(* IEC 61131-3 sources: volt/packages/volt-lsp-iec/test-corpus/pro2193/Device/Plc Logic/Application/99 Library/Function Blocks/Sensors, 4 files *)

(* ---- DigitalSensorFB.pou ---- *)
// Basic FB for a digital sensor, adds invert functionality
{attribute 'no_explicit_call' := 'No need to call this FB. No code to execute!'}
{attribute 'symbol' := 'none'}
{attribute 'monitoring_display' := 'IsActive'}
FUNCTION_BLOCK DigitalSensorFB
IMPLEMENTS IDigitalSensor
VAR_INPUT
	{attribute 'symbol' := 'read'}		sensorInput		: BOOL;
END_VAR
VAR
	_isInverted		: BOOL;
END_VAR

%LANGUAGE ST

END_FUNCTION_BLOCK

// FB_Init is always available implicitly and it is used primarily for initialization.
// The return value is not evaluated. For a specific influence, you can also declare the
// methods explicitly and provide additional code there with the standard initialization
// code. You can evaluate the return value.
{attribute 'hide'}
METHOD FB_Init: BOOL
VAR_INPUT
	bInitRetains: BOOL; // TRUE: the retain variables are initialized (reset warm / reset cold)
	bInCopyCode: BOOL;  // TRUE: the instance will be copied to the copy code afterward (online change)

	invert			: BOOL;	// Sensor or photocell signal should be inverted
END_VAR

%LANGUAGE ST
_isInverted := invert;

END_METHOD

// Sensor is active (SensorInput is opposite of the Invert signal)
{attribute 'monitoring':='call'}
PROPERTY IsActive : BOOL

GET
PUBLIC
VAR
END_VAR

%LANGUAGE ST
IsActive := SensorInput = NOT _isInverted;

END_GET
END_PROPERTY

// Sensor is inactive (SensorInput is false (or true when inverted))
{attribute 'monitoring':='call'}
PROPERTY IsInactive : BOOL

GET
PUBLIC
VAR
END_VAR

%LANGUAGE ST
IsInactive := NOT IsActive;

END_GET
END_PROPERTY

(* ---- DigitalSensorWithEnableFB.pou ---- *)
// When disabled a sensor will always return TRUE when asked! So the program will continue and ignore the sensor.
{attribute 'no_explicit_call' := 'No need to call this FB. No code to execute!'}
{attribute 'symbol' := 'none'}
{attribute 'monitoring_display' := 'IsActive'}
FUNCTION_BLOCK DigitalSensorWithEnableFB
EXTENDS DigitalSensorFB
VAR
	_isEnabled		: BOOL;
END_VAR

%LANGUAGE ST

END_FUNCTION_BLOCK

// Sensor is active (SensorInput is opposite of the Invert signal)
{attribute 'monitoring':='call'}
PROPERTY IsActive : BOOL

GET
PUBLIC
VAR
END_VAR

%LANGUAGE ST
IsActive := NOT IsEnabled OR_ELSE SUPER^.IsActive;

END_GET
END_PROPERTY

// Sensor is enabled or disabled
{attribute 'monitoring':='call'}
PROPERTY IsEnabled : BOOL

GET
PUBLIC
VAR
END_VAR

%LANGUAGE ST
IsEnabled := _isEnabled;

END_GET
SET
PUBLIC
VAR
END_VAR

%LANGUAGE ST
_isEnabled := IsEnabled;

END_SET
END_PROPERTY

// Sensor is inactive (SensorInput is false (or true when inverted))
{attribute 'monitoring':='call'}
PROPERTY IsInactive : BOOL

GET
PUBLIC
VAR
END_VAR

%LANGUAGE ST
IsInactive := NOT IsEnabled OR_ELSE SUPER^.IsInactive;

END_GET
END_PROPERTY

(* ---- DigitalSensorWithTriggersAndTimeoutFB.pou ---- *)
// Add timeout alarm to a digital input (remember to call IsInactive method when signal should be FALSE!)
{attribute 'symbol' := 'none'}
{attribute 'monitoring_display' := 'IsActive'}
FUNCTION_BLOCK DigitalSensorWithTriggersAndTimeoutFB
EXTENDS DigitalSensorWithTriggersFB
VAR_INPUT
	Pt					: REAL	:= 5;	// Time to pass (in sec.), after which the alarm trips.
END_VAR
VAR_OUTPUT
	alarmActive			: BOOL;			// High when input is not TRUE or FALSE within the given timeout
END_VAR
VAR
	SignalTimeout		: SignalTimeoutFB;
END_VAR

%LANGUAGE ST
SUPER^();

SignalTimeout(
	timeOut		:= Pt,
	input		:= SensorInput = NOT _isInverted,
	alarmActive	=> alarmActive);

END_FUNCTION_BLOCK

// Sensor is active (Enable is high and SensorInput is opposite of the Invert signal)
{attribute 'monitoring':='variable'}
PROPERTY IsActive : BOOL

GET
PUBLIC
VAR
END_VAR

%LANGUAGE ST
IsActive := SignalTimeout.GetValue(TRUE);

END_GET
END_PROPERTY

// Sensor is active (Enable is high and SensorInput is opposite of the Invert signal)
{attribute 'monitoring':='variable'}
PROPERTY IsInactive : BOOL

GET
PUBLIC
VAR
END_VAR

%LANGUAGE ST
IsInactive := SignalTimeout.GetValue(FALSE);

END_GET
END_PROPERTY

(* ---- DigitalSensorWithTriggersFB.pou ---- *)
// Add rising and falling trigger to a digital input (remember to call the instance of this FB!)
{attribute 'symbol' := 'none'}
{attribute 'monitoring_display' := 'IsActive'}
FUNCTION_BLOCK DigitalSensorWithTriggersFB
EXTENDS DigitalSensorFB
VAR
	Trigger			: TriggerFB;
END_VAR

%LANGUAGE ST
Trigger.Call(CLK := SensorInput = NOT _isInverted);

END_FUNCTION_BLOCK

PROPERTY Falling : BOOL

GET
PUBLIC
VAR
END_VAR

%LANGUAGE ST
Falling := Trigger.Q_Falling;

END_GET
END_PROPERTY

PROPERTY Rising : BOOL

GET
PUBLIC
VAR
END_VAR

%LANGUAGE ST
Rising := Trigger.Q_Rising;

END_GET
END_PROPERTY
